Yaskawa INFORM job: long_pipe_hz_cylinder_program.JBI

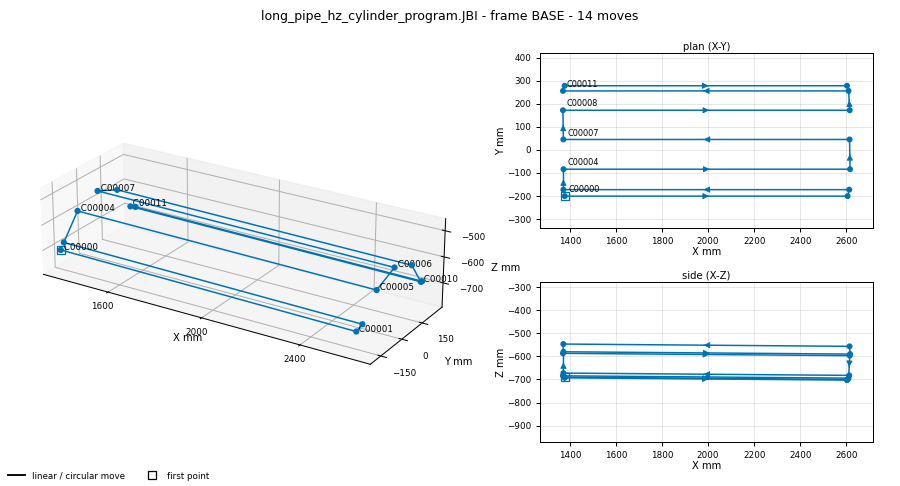
[picture p0: tool path of long_pipe_hz_cylinder_program.JBI in frame BASE, 14 of 17 moves have a stored position in this frame; points joined in program order, loops and branches not executed]
/JOB
//NAME long_pipe_hz_cylinder_program
//POS
///NPOS 14,0,14,0,0,0
///TOOL 0
///POSTYPE BASE
///RECTAN
///RCONF 0,0,0,0,0,0,0,0,0,0,0,0,0,0,0,0,0,0,0,0,0,0,0,0
C00000=1378.152390,-200.495114,-689.902054,175.000000,-83.878792,90.049349
C00001=2605.056971,-200.496124,-699.765099,175.000000,-83.878792,90.049349
C00002=2612.246983,-172.305896,-682.233930,-175.000000,-61.681524,90.248152
C00003=1372.083338,-172.304875,-672.264296,-175.000000,-61.681524,90.248152
C00004=1372.591829,-83.625199,-579.823095,175.000000,-30.702822,90.775626
C00005=2615.559308,-83.626221,-589.815269,175.000000,-30.702822,90.775626
C00006=2613.517615,45.345749,-556.277428,175.000000,5.000000,-5.000000
C00007=1371.816165,45.346770,-546.295432,175.000000,5.000000,-5.000000
C00008=1370.223285,172.107365,-586.651457,175.000000,-33.769906,-90.688881
C00009=2614.308682,172.106341,-596.652618,175.000000,-33.769906,-90.688881
C00010=2609.225187,255.942978,-694.160688,-175.000000,-64.878346,-90.216020
C00011=1370.276846,255.943998,-684.200823,-175.000000,-64.878346,-90.216020
C00012=1377.559331,278.386258,-692.858533,175.000000,-85.775267,-90.034071
C00013=2602.278755,278.385251,-702.704012,175.000000,-60.000000,-90.034071
///POSTYPE PULSE
///PULSE
EX00000=270336.0
///POSTYPE PULSE
///PULSE
EC00000=270336.0
EC00001=270336.0
EC00002=270336.0
EC00003=270336.0
EC00004=270336.0
EC00005=270336.0
EC00006=270336.0
EC00007=270336.0
EC00008=270336.0
EC00009=270336.0
EC00010=270336.0
EC00011=270336.0
EC00012=270336.0
EC00013=270336.0
//INST
///DATE 2023/08/15 13:30
///ATTR SC,RW,RJ
////FRAME BASE
///GROUP1 RB1,ST1
NOP
MOVJ P009 EX000 VJ=15.00
MOVJ C00000 EC00000 VJ=15.0
CALL JOB:SPYON
MOVL C00001 EC00001 V=150.0
MOVL C00002 EC00002 V=150.0
MOVL C00003 EC00003 V=150.0
MOVL C00004 EC00004 V=150.0
MOVL C00005 EC00005 V=150.0
MOVL C00006 EC00006 V=150.0
MOVL C00007 EC00007 V=150.0
MOVL C00008 EC00008 V=150.0
MOVL C00009 EC00009 V=150.0
MOVL C00010 EC00010 V=150.0
MOVL C00011 EC00011 V=150.0
MOVL C00012 EC00012 V=150.0
MOVL C00013 EC00013 V=150.0
CALL JOB:SPYOF
MOVJ P009 VJ=15.00
MOVL P009 EX00000 V=150.0
END
